// TIA Portal V17 export
// export: Created 2023-12-22T15:08:02.6117163Z, ExportSetting WithDefaults, DisplayName Totally Integrated Automation Portal, DisplayVersion V17, DisplayName TIA Portal Openness, DisplayVersion V17, DisplayName TIA Portal Version Control Interface, DisplayVersion V17, DisplayName STEP 7 Professional, DisplayVersion V17, DisplayName STEP 7 Safety, DisplayVersion V17, DisplayName WinCC Advanced, DisplayVersion V17
FUNCTION_BLOCK "AIx"   // FB220, LAD
{ S7_Optimized_Access := 'FALSE' }
VERSION : 0.1
// Signal - PIW код сигнала от датчика
// pulse - частота алгоритма фильтрации
// Result - результат обработки сигнала, формат Real
// stored: AutoNumber false, IsIECCheckEnabled false, SetENOAutomatically false, UDAEnableTagReadback false
   VAR DB_SPECIFIC
      Time_DTL { S7_SetPoint := 'True'} : DTL;
   END_VAR
   VAR_TEMP   // added for the SCL form of the ladder/FBD networks
      _w1 : Bool;
   END_VAR
BEGIN

REGION Network 1: Датчик давления 1 - 2
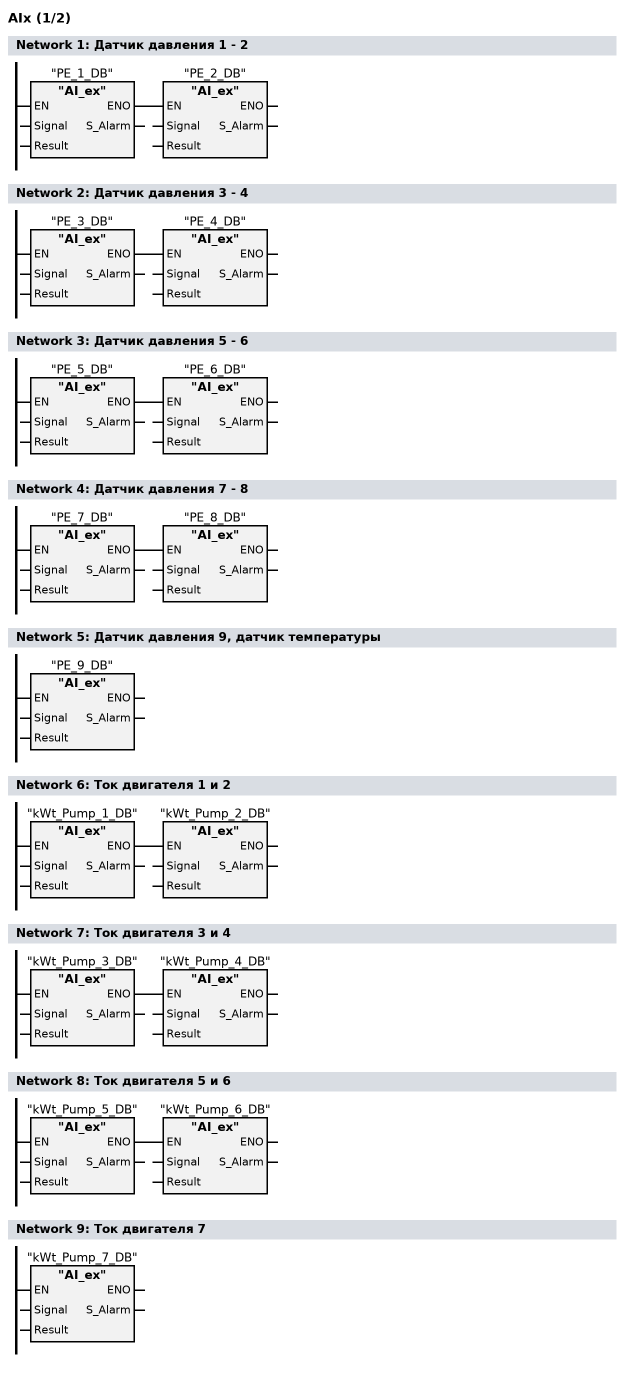
   RUNG wire#powerrail
      "PE_1_DB"(Signal :=, Result :=, S_Alarm =>)
      "PE_2_DB"(Signal :=, Result :=, S_Alarm =>)
   END_RUNG
   // the same network as SCL:
   "PE_1_DB"(ENO => #_w1);   // "AI_ex"
   IF #_w1 THEN
       "PE_2_DB"();   // "AI_ex"
   END_IF;
END_REGION

REGION Network 2: Датчик давления 3 - 4
   RUNG wire#powerrail
      "PE_3_DB"(Signal :=, Result :=, S_Alarm =>)
      "PE_4_DB"(Signal :=, Result :=, S_Alarm =>)
   END_RUNG
   // the same network as SCL:
   "PE_3_DB"(ENO => #_w1);   // "AI_ex"
   IF #_w1 THEN
       "PE_4_DB"();   // "AI_ex"
   END_IF;
END_REGION

REGION Network 3: Датчик давления 5 - 6
   RUNG wire#powerrail
      "PE_5_DB"(Signal :=, Result :=, S_Alarm =>)
      "PE_6_DB"(Signal :=, Result :=, S_Alarm =>)
   END_RUNG
   // the same network as SCL:
   "PE_5_DB"(ENO => #_w1);   // "AI_ex"
   IF #_w1 THEN
       "PE_6_DB"();   // "AI_ex"
   END_IF;
END_REGION

REGION Network 4: Датчик давления 7 - 8
   RUNG wire#powerrail
      "PE_7_DB"(Signal :=, Result :=, S_Alarm =>)
      "PE_8_DB"(Signal :=, Result :=, S_Alarm =>)
   END_RUNG
   // the same network as SCL:
   "PE_7_DB"(ENO => #_w1);   // "AI_ex"
   IF #_w1 THEN
       "PE_8_DB"();   // "AI_ex"
   END_IF;
END_REGION

REGION Network 5: Датчик давления 9, датчик температуры
   RUNG wire#powerrail
      "PE_9_DB"(Signal :=, Result :=, S_Alarm =>)
   END_RUNG
   // the same network as SCL:
   "PE_9_DB"();   // "AI_ex"
END_REGION

REGION Network 6: Ток двигателя 1 и 2
   RUNG wire#powerrail
      "kWt_Pump_1_DB"(Signal :=, Result :=, S_Alarm =>)
      "kWt_Pump_2_DB"(Signal :=, Result :=, S_Alarm =>)
   END_RUNG
   // the same network as SCL:
   "kWt_Pump_1_DB"(ENO => #_w1);   // "AI_ex"
   IF #_w1 THEN
       "kWt_Pump_2_DB"();   // "AI_ex"
   END_IF;
END_REGION

REGION Network 7: Ток двигателя 3 и 4
   RUNG wire#powerrail
      "kWt_Pump_3_DB"(Signal :=, Result :=, S_Alarm =>)
      "kWt_Pump_4_DB"(Signal :=, Result :=, S_Alarm =>)
   END_RUNG
   // the same network as SCL:
   "kWt_Pump_3_DB"(ENO => #_w1);   // "AI_ex"
   IF #_w1 THEN
       "kWt_Pump_4_DB"();   // "AI_ex"
   END_IF;
END_REGION

REGION Network 8: Ток двигателя 5 и 6
   RUNG wire#powerrail
      "kWt_Pump_5_DB"(Signal :=, Result :=, S_Alarm =>)
      "kWt_Pump_6_DB"(Signal :=, Result :=, S_Alarm =>)
   END_RUNG
   // the same network as SCL:
   "kWt_Pump_5_DB"(ENO => #_w1);   // "AI_ex"
   IF #_w1 THEN
       "kWt_Pump_6_DB"();   // "AI_ex"
   END_IF;
END_REGION

REGION Network 9: Ток двигателя 7
   RUNG wire#powerrail
      "kWt_Pump_7_DB"(Signal :=, Result :=, S_Alarm =>)
   END_RUNG
   // the same network as SCL:
   "kWt_Pump_7_DB"();   // "AI_ex"
END_REGION

REGION Network 10
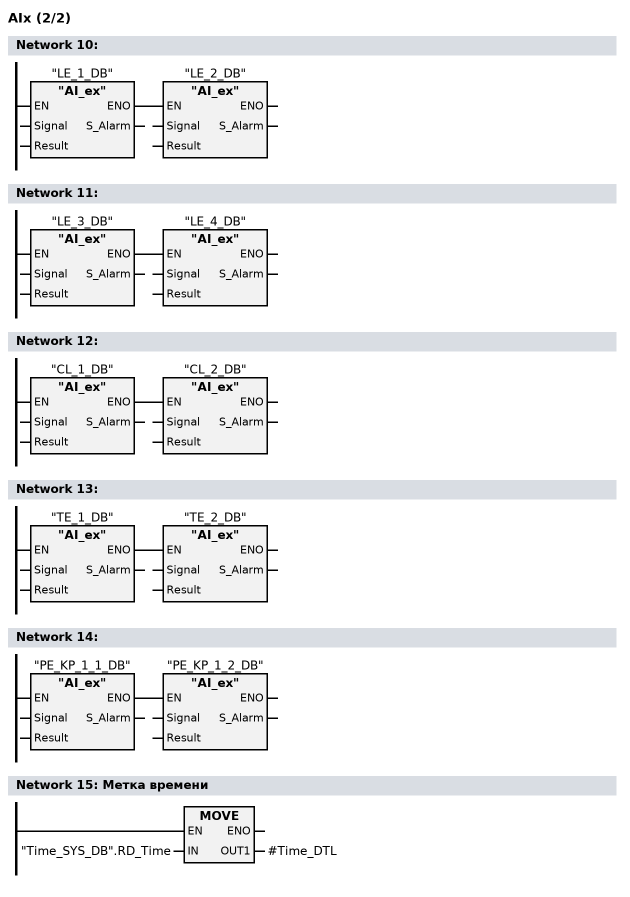
   RUNG wire#powerrail
      "LE_1_DB"(Signal :=, Result :=, S_Alarm =>)
      "LE_2_DB"(Signal :=, Result :=, S_Alarm =>)
   END_RUNG
   // the same network as SCL:
   "LE_1_DB"(ENO => #_w1);   // "AI_ex"
   IF #_w1 THEN
       "LE_2_DB"();   // "AI_ex"
   END_IF;
END_REGION

REGION Network 11
   RUNG wire#powerrail
      "LE_3_DB"(Signal :=, Result :=, S_Alarm =>)
      "LE_4_DB"(Signal :=, Result :=, S_Alarm =>)
   END_RUNG
   // the same network as SCL:
   "LE_3_DB"(ENO => #_w1);   // "AI_ex"
   IF #_w1 THEN
       "LE_4_DB"();   // "AI_ex"
   END_IF;
END_REGION

REGION Network 12
   RUNG wire#powerrail
      "CL_1_DB"(Signal :=, Result :=, S_Alarm =>)
      "CL_2_DB"(Signal :=, Result :=, S_Alarm =>)
   END_RUNG
   // the same network as SCL:
   "CL_1_DB"(ENO => #_w1);   // "AI_ex"
   IF #_w1 THEN
       "CL_2_DB"();   // "AI_ex"
   END_IF;
END_REGION

REGION Network 13
   RUNG wire#powerrail
      "TE_1_DB"(Signal :=, Result :=, S_Alarm =>)
      "TE_2_DB"(Signal :=, Result :=, S_Alarm =>)
   END_RUNG
   // the same network as SCL:
   "TE_1_DB"(ENO => #_w1);   // "AI_ex"
   IF #_w1 THEN
       "TE_2_DB"();   // "AI_ex"
   END_IF;
END_REGION

REGION Network 14
   RUNG wire#powerrail
      "PE_KP_1_1_DB"(Signal :=, Result :=, S_Alarm =>)
      "PE_KP_1_2_DB"(Signal :=, Result :=, S_Alarm =>)
   END_RUNG
   // the same network as SCL:
   "PE_KP_1_1_DB"(ENO => #_w1);   // "AI_ex"
   IF #_w1 THEN
       "PE_KP_1_2_DB"();   // "AI_ex"
   END_IF;
END_REGION

REGION Network 15: Метка времени
   RUNG wire#powerrail
      Move(in := "Time_SYS_DB".RD_Time, out1 => #Time_DTL)
   END_RUNG
   // the same network as SCL:
   #Time_DTL := "Time_SYS_DB".RD_Time;
END_REGION
END_FUNCTION_BLOCK
